Staubli VAL3: extractPos.pgx

public program extractPos(string x_sInString, string x_sBreakChar, num& x_nVal1[], num& x_nVal2[])
  local bool l_bOk
begin
  // This program extracts 2 numerical values from the input string
  //
  // Input Param
  //  x_sInstring     : Input string which contains the values to extract
  //  x_sBreakChar    : Break character
  //
  // Output Param
  //  x_nVal1                  : First numerical value
  //  x_nVal2                  : Second numerical value
  //
  // Created 15/01/01                              C.CURRIVAND
  //---------------------------------------------------------
  x_sInString=toNum(x_sInString,x_nVal1,l_bOk)
  x_sInString=toNum(x_sInString,x_nVal2,l_bOk)
end
